Universal Robots PolyScope program: pinacolada.urp

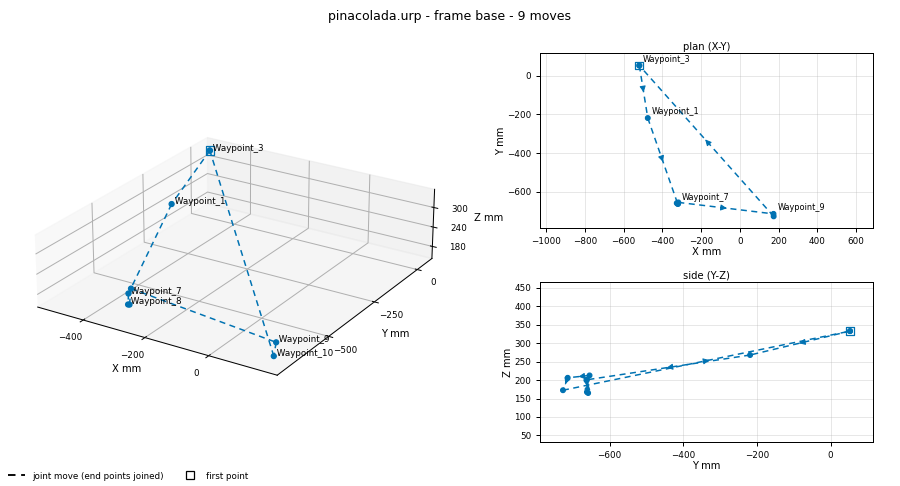
[picture p0: tool path of pinacolada.urp in frame base, 9 of 9 moves have a stored position in this frame; points joined in program order, loops and branches not executed]
Program pinacolada (installation=default directory=/programs/AronLauschOrdering createdIn=5.12.6.1102099 lastSavedIn=5.12.6.1102099 robotSerialNumber=20215500597)
Calibrated DH parameters: a=[0.000193, -0.066673, -0.391568, -0.000012, 0.00005, 0]; d=[0.162643, -472.05677, 465.132521, 7.058239, 0.099746, 0.099582]; alpha=[1.571116, 0.00089, 0.003862, 1.569269, -1.569248, 0]; deltaTheta=[0, -1.413394, 7.628392, 0.068187, 0, -0.000001]
Robot Program (runOnlyOnce=true)
  MoveJ speed 60 deg/s, acceleration 80 deg/s^2 (useActiveTCP=true) feature=Base
    Waypoint Waypoint_3: TCP in base x=-519.145 y=52.76 z=332.958 mm, rx=-3.1405 ry=-0.0837 rz=0.0002 rad; joints [-20.664, -88.123, 82.733, -84.528, -89.812, 66.326] deg; TCP offset x=0 y=0 z=191.5 mm, rx=0 ry=0 rz=0 rad
  MoveJ speed 60 deg/s, acceleration 80 deg/s^2 (useActiveTCP=true) feature=Base
    Waypoint Waypoint_1: TCP in base x=-475.505 y=-218.538 z=268.037 mm, rx=-2.9452 ry=1.0885 rz=-0.005 rad; joints [9.852, -87.863, 91.897, -93.738, -89.803, 140.495] deg
  MoveJ speed 60 deg/s, acceleration 80 deg/s^2 (useActiveTCP=true) feature=Base
    Waypoint Waypoint_7: TCP in base x=-320.581 y=-662.671 z=200.67 mm, rx=-3.1402 ry=-0.0898 rz=-0.0001 rad; joints [53.721, -56.831, 60.673, -93.747, -89.799, 140.497] deg; TCP offset x=0 y=0 z=191.5 mm, rx=0 ry=0 rz=0 rad
    URCap Gripper (Robotiq_Grippers, Robotiq Inc.) dataModel(position=0.0, force=100.0, speed=100.0, positionInDouble=0.0, forceInDouble=100.0, speedInDouble=100.0, slaveIds=[9], blocking=true)
    Waypoint Waypoint_8: TCP in base x=-325.774 y=-658.115 z=164.889 mm, rx=-3.1407 ry=-0.0744 rz=0 rad; joints [53.172, -56.504, 65.409, -98.814, -89.8, 140.53] deg; TCP offset x=0 y=0 z=191.5 mm, rx=0 ry=0 rz=0 rad
    Waypoint Waypoint_down: TCP in base x=-318.84 y=-661.414 z=167.597 mm, rx=-3.0845 ry=-0.1578 rz=-0.0097 rad; joints [54.422, -54.45, 61.076, -93.935, -91.408, 138.656] deg
    URCap Gripper (Robotiq_Grippers, Robotiq Inc.) dataModel(position=100.0, force=100.0, speed=100.0, positionInDouble=100.0, forceInDouble=100.0, speedInDouble=100.0, slaveIds=[9], blocking=true)
    Waypoint Waypoint_up: TCP in base x=-317.689 y=-654.317 z=212.673 mm, rx=-3.114 ry=-0.157 rz=0.0451 rad; joints [54.377, -58.01, 60.813, -92.699, -91.928, 138.658] deg
    Waypoint Waypoint_9: TCP in base x=173.955 y=-713.606 z=206.243 mm, rx=-2.1501 ry=-2.2722 rz=0.0499 rad; joints [93.957, -57.415, 60.987, -94.172, -91.646, 90.839] deg
    Waypoint Waypoint_10: TCP in base x=174.863 y=-726.44 z=172.474 mm, rx=-2.2338 ry=-2.2004 rz=-0.0016 rad; joints [93.3, -54.466, 60.914, -96.064, -89.981, 94.225] deg
    URCap Gripper (Robotiq_Grippers, Robotiq Inc.) dataModel(position=0.0, force=100.0, speed=100.0, positionInDouble=0.0, forceInDouble=100.0, speedInDouble=100.0, slaveIds=[9], blocking=true)
    Waypoint Waypoint_3: TCP in base x=-519.145 y=52.76 z=332.958 mm, rx=-3.1405 ry=-0.0837 rz=0.0002 rad; joints [-20.664, -88.123, 82.733, -84.528, -89.812, 66.326] deg
